INTERFACE I_BaseUnit EXTENDS __SYSTEM.IQueryInterface

END_INTERFACE

(* stored: Version 1.1.0.1, ProductVersion 3.1.4026.18
   Itf I_BaseUnit: Id {318f29b4-8873-4aee-b299-1602a6e50df3} *)
